Yaskawa INFORM job: N_R2_D34(P)(-165,-90).JBI

/JOB
//NAME N_R2_D34(P)(-165,-90)
//POS
///NPOS 212,212,212,10,0,0
///TOOL 0
///POSTYPE PULSE
///PULSE
C00000=-39723,-76225,-106677,19950,71807,76871
C00001=-136716,-73683,-105524,19345,72156,77265
C00002=-161407,-91524,-110310,15012,103390,71507
C00003=-108598,-106188,-63612,3932,70077,81231
C00004=-108146,-105032,-58861,3973,67731,81309
C00005=-107957,-104486,-56911,3991,66805,81343
C00006=-107899,-103124,-54603,4010,66084,81338
C00007=-107918,-103337,-55008,4006,66224,81336
C00008=-107946,-103390,-55013,4008,66201,81326
C00009=-107540,-105489,-55732,4011,65548,81444
C00010=-107946,-103390,-55013,4008,66201,81326
C00011=-108136,-103965,-56983,3989,67125,81292
C00012=-108589,-105196,-61782,3946,69462,81214
C00013=-104387,-140393,-91773,2539,65045,84360
C00014=-108543,-122383,-87788,3041,71761,81393
C00015=-108190,-121281,-83186,3043,69485,81459
C00016=-108044,-120747,-81302,3044,68596,81488
C00017=-107986,-119544,-79172,3051,67902,81491
C00018=-108002,-119703,-79496,3051,68020,81488
C00019=-108060,-119698,-79501,3057,68028,81468
C00020=-107657,-122309,-80316,3030,67174,81589
C00021=-108060,-119698,-79501,3057,68028,81468
C00022=-108206,-120261,-81401,3055,68912,81439
C00023=-108559,-121443,-86043,3052,71171,81373
C00024=-104043,-152650,-104301,-20,47297,80621
C00025=-107961,-134888,-100622,1830,53982,78996
C00026=-108046,-130238,-95035,1891,52935,78942
C00027=-108079,-128417,-92795,1916,52493,78920
C00028=-108021,-127286,-90730,1909,51803,78931
C00029=-108035,-127446,-91054,1912,51920,78927
C00030=-108130,-127490,-91067,1954,51908,78887
C00031=-107729,-130486,-91965,1802,50912,79038
C00032=-108130,-127490,-91067,1954,51908,78887
C00033=-108097,-129313,-93314,1928,52353,78910
C00034=-108012,-133964,-98916,1865,53408,78964
C00035=-177548,-171463,-116071,22976,53227,57999
C00036=-173065,-131414,-104138,1882,83052,64081
C00037=-174658,-131451,-100095,1929,80584,63502
C00038=-175319,-131311,-98421,1949,79642,63262
C00039=-175466,-130194,-96381,1956,78964,63202
C00040=-175319,-131311,-98421,1949,79642,63262
C00041=-175487,-130273,-96656,1956,79094,63196
C00042=-177055,-132761,-97424,1996,78327,62650
C00043=-175487,-130273,-96656,1956,79094,63196
C00044=-174824,-130456,-98346,1936,80024,63437
C00045=-173224,-130544,-102436,1888,82455,64018
C00046=-183578,-145461,-102579,23161,59534,56897
C00047=-173554,-122008,-87484,5289,73895,63503
C00048=-174753,-120461,-82756,5436,71868,62996
C00049=-175245,-119759,-80826,5498,71077,62789
C00050=-175392,-118530,-78687,5530,70405,62707
C00051=-175367,-118686,-78973,5525,70498,62719
C00052=-175370,-118724,-79021,5525,70509,62719
C00053=-176937,-120728,-79681,5662,69994,62147
C00054=-175370,-118724,-79021,5525,70509,62719
C00055=-174875,-119452,-80967,5462,71295,62928
C00056=-173672,-121073,-85733,5313,73308,63437
C00057=-178684,-130472,-89403,5463,71088,61622
C00058=-172855,-106156,-63418,1950,70986,63967
C00059=-174444,-104513,-58519,2015,68854,63388
C00060=-175103,-103777,-56512,2042,68014,63147
C00061=-175249,-102388,-54194,2055,67305,63085
C00062=-175217,-102613,-54582,2053,67427,63098
C00063=-175253,-102649,-54567,2054,67400,63085
C00064=-176818,-104272,-55156,2098,66967,62541
C00065=-175253,-102649,-54567,2054,67400,63085
C00066=-174591,-103412,-56593,2026,68239,63327
C00067=-172994,-105125,-61540,1961,70363,63910
C00068=-156260,-82084,-105549,20460,72443,69801
C00069=-137260,-84248,-120477,10166,77039,76481
C00070=-137260,-138866,-129024,10166,31486,76481
C00071=-31464,-162597,-129024,10166,12061,76481
C00072=11401,-148032,-125424,11666,35639,75770
C00073=126224,-114648,-117374,36487,17100,65054
C00074=135046,-120043,-103653,15284,86568,49617
C00075=106845,-105753,-62932,583,70286,77102
C00076=106393,-104585,-58171,607,67960,76935
C00077=106203,-104034,-56217,618,67041,76865
C00078=106162,-102674,-53905,622,66318,76847
C00079=106166,-102878,-54243,622,66421,76849
C00080=106334,-102921,-54287,616,66425,76907
C00081=105882,-105004,-55005,634,65800,76748
C00082=106334,-102921,-54287,616,66425,76907
C00083=106522,-103500,-56261,605,67341,76976
C00084=106972,-104744,-61071,581,69658,77143
C00085=104601,-139074,-91382,1569,66028,76192
C00086=106568,-121926,-87059,1557,71993,76932
C00087=106224,-120810,-82448,1613,69736,76782
C00088=106082,-120272,-80560,1636,68854,76720
C00089=106040,-119071,-78428,1648,68159,76695
C00090=106046,-119261,-78757,1646,68265,76699
C00091=106190,-119319,-78791,1631,68253,76749
C00092=105732,-121900,-79600,1688,67434,76576
C00093=106190,-119319,-78791,1631,68253,76749
C00094=106332,-119888,-80695,1608,69129,76811
C00095=106675,-121089,-85348,1552,71368,76961
C00096=103496,-155225,-104630,7919,46945,74289
C00097=105785,-134375,-99806,6437,54295,75766
C00098=105945,-129762,-94221,6456,53222,75764
C00099=106008,-127954,-91981,6467,52771,75762
C00100=105966,-126823,-89914,6544,52087,75701
C00101=105978,-126937,-90184,6529,52194,75712
C00102=106125,-127008,-90229,6468,52174,75772
C00103=105664,-129959,-91118,6752,51247,75517
C00104=106125,-127008,-90229,6468,52174,75772
C00105=106062,-128819,-92476,6456,52628,75775
C00106=105903,-133434,-98077,6434,53709,75777
C00107=128132,-113142,-93523,-3473,64221,79775
C00108=127541,-110622,-88467,-3323,62383,79607
C00109=127305,-109564,-86417,-3263,61656,79539
C00110=127138,-106637,-85321,-3181,62477,79452
C00111=127288,-110024,-87846,-3238,62297,79514
C00112=123322,-109914,-86529,-1878,61418,78027
C00113=118008,-109912,-86522,-16,61352,76001
C00114=114024,-109560,-86400,1379,61491,74484
C00115=114240,-110677,-88470,1295,62187,74574
C00116=114784,-113359,-93579,1090,63945,74797
C00117=120605,-145695,-100878,-6504,46630,80491
C00118=128077,-118688,-85011,-1726,71284,79523
C00119=126726,-104779,-76666,-1004,79571,78924
C00120=126488,-104947,-74265,-1002,78005,78856
C00121=126338,-102371,-73283,-996,78722,78799
C00122=126472,-105599,-75792,-1000,78609,78846
C00123=122432,-105195,-74343,-890,77878,77473
C00124=117012,-105110,-74308,-735,77846,75625
C00125=112968,-104735,-74177,-617,77924,74245
C00126=113438,-104642,-76602,-628,79468,74397
C00127=113371,-116037,-84290,-102,73201,74367
C00128=120594,-140938,-90128,-5435,60827,78775
C00129=125790,-88282,-54907,-1855,89205,80575
C00130=125481,-89790,-51762,-1908,86488,80513
C00131=125349,-90285,-50434,-1932,85415,80486
C00132=125231,-88136,-49532,-1951,85961,80439
C00133=125335,-91126,-52116,-1933,86017,80473
C00134=121365,-90427,-50480,-2603,85262,79186
C00135=116055,-90283,-50421,-3488,85105,77452
C00136=119868,-90564,-50050,-7604,84693,77985
C00137=120335,-90112,-51383,-7520,85779,78074
C00138=121427,-88708,-54542,-7332,88521,78274
C00139=128084,-118876,-109490,15608,91937,64784
C00140=126224,-114648,-117374,36487,17100,65054
C00141=118781,-153852,-129024,32591,23356,65054
C00142=12469,-167082,-125424,11666,16324,75770
C00143=-137258,-84249,-120477,10166,64820,76481
C00144=-160540,-100856,-113062,23154,68828,67580
C00145=-129704,-123203,-96216,9710,57100,77822
C00146=-128351,-111854,-90022,8241,62769,78816
C00147=-127965,-110264,-86953,8187,61668,78883
C00148=-127962,-110732,-88383,8139,62302,78931
C00149=-127784,-107324,-85860,8064,62480,79012
C00150=-123964,-110663,-87100,6807,61182,80388
C00151=-118738,-110727,-87139,4953,60792,82376
C00152=-114730,-110424,-87053,3503,60683,83913
C00153=-115087,-112114,-90154,3597,61737,83810
C00154=-115034,-127353,-96665,3487,52332,83552
C00155=-120587,-140955,-100514,6147,49960,81085
C00156=-130219,-122449,-86471,8825,68877,76131
C00157=-128194,-104501,-77199,7275,80206,77627
C00158=-127952,-104717,-74821,7301,78623,77617
C00159=-127948,-105352,-76341,7288,79227,77654
C00160=-127769,-102129,-73832,7281,79322,77721
C00161=-123925,-105065,-74954,7196,78166,78974
C00162=-118667,-105119,-74990,7025,77701,80756
C00163=-114634,-104852,-74915,6870,77446,82130
C00164=-115105,-104718,-77320,6855,79024,82055
C00165=-115436,-113024,-84089,6687,75142,81750
C00166=-120582,-141029,-90717,5476,61131,81670
C00167=-128285,-87656,-54320,10457,89548,79035
C00168=-127487,-89201,-51235,10596,86798,79071
C00169=-127146,-89710,-49931,10663,85708,79092
C00170=-127144,-90552,-51616,10658,86302,79143
C00171=-126986,-87570,-49030,10686,86223,79189
C00172=-123182,-89955,-50036,11339,85127,80359
C00173=-118012,-89954,-50056,12180,84414,82017
C00174=-114050,-89707,-49981,12789,83904,83291
C00175=-114638,-89281,-51315,12685,85009,83208
C00176=-116016,-87939,-54478,12458,87793,83023
C00177=-137088,-110527,-71299,-11812,85392,74901
C00178=-151248,-92745,-56294,-13309,83013,70315
C00179=-153775,-93208,-52742,-13646,80246,69760
C00180=-154842,-93280,-51259,-13793,79148,69522
C00181=-153977,-91331,-50464,-13683,79788,69743
C00182=-154783,-94178,-52960,-13764,79728,69477
C00183=-158502,-91409,-50586,-14135,79075,68289
C00184=-162995,-88717,-49588,-14508,79057,66760
C00185=-166247,-86464,-48726,-14744,79098,65642
C00186=-165114,-86470,-50212,-14620,80180,65901
C00187=-162400,-86203,-53771,-14331,82909,66512
C00188=-168399,-109053,-82349,-2367,78378,65064
C00189=-153094,-88623,-71084,-2982,100007,61638
C00190=-154899,-90939,-68502,-3287,97162,61087
C00191=-155658,-91729,-67395,-3417,96045,60858
C00192=-154888,-89489,-66414,-3281,96623,61105
C00193=-155605,-92249,-68886,-3413,96696,60858
C00194=-158825,-89499,-66505,-3999,96496,59762
C00195=-162743,-86354,-65215,-4713,97104,58398
C00196=-165600,-83764,-64121,-5229,97582,57396
C00197=-164765,-83025,-65209,-5099,98681,57638
C00198=-162766,-80848,-67746,-4792,101474,58222
C00199=-167065,-111844,-93662,10716,66234,64857
C00200=-163867,-82906,-82329,-2559,109140,68035
C00201=-165085,-87347,-80821,-2728,105894,67672
C00202=-165597,-88966,-80125,-2801,104618,67519
C00203=-165533,-89090,-81425,-2801,105355,67525
C00204=-164697,-86621,-79049,-2646,105191,67825
C00205=-162740,-91967,-81360,-2276,103927,68542
C00206=-158823,-95635,-82824,-1559,103037,69935
C00207=-155656,-98251,-83839,-981,102367,71052
C00208=-155268,-96625,-84596,-916,103674,71178
C00209=-154353,-92138,-86254,-764,107009,71479
C00210=-136716,-73683,-105524,19345,72156,77265
C00211=-39723,-76225,-106677,19950,71807,76871
BC00000=295325,674563,1075175
BC00001=353535,895977,1075175
BC00002=353535,975867,1075175
BC00003=342454,1030449,1075175
BC00004=342454,1030449,1075175
BC00005=342454,1030449,1075175
BC00006=342454,1030449,1075175
BC00007=342454,1030449,1075175
BC00008=342454,1030449,1075175
BC00009=342454,1030449,1075175
BC00010=342454,1030449,1075175
BC00011=342454,1030449,1075175
BC00012=342454,1030449,1075175
BC00013=342372,1053588,1075175
BC00014=342372,1053588,1075175
BC00015=342372,1053588,1075175
BC00016=342372,1053588,1075175
BC00017=342372,1053588,1075175
BC00018=342372,1053588,1075175
BC00019=342372,1053588,1075175
BC00020=342372,1053588,1075175
BC00021=342372,1053588,1075175
BC00022=342372,1053588,1075175
BC00023=342372,1053588,1075175
BC00024=339313,1046331,1075175
BC00025=339313,1046331,1075175
BC00026=339313,1046331,1075175
BC00027=339313,1046331,1075175
BC00028=339313,1046331,1075175
BC00029=339313,1046331,1075175
BC00030=339313,1046331,1075175
BC00031=339313,1046331,1075175
BC00032=339313,1046331,1075175
BC00033=339313,1046331,1075175
BC00034=339313,1046331,1075175
BC00035=316444,1061550,1075175
BC00036=316336,1108016,1075175
BC00037=316336,1108016,1075175
BC00038=316336,1108016,1075175
BC00039=316336,1108016,1075175
BC00040=316336,1108016,1075175
BC00041=316336,1108016,1075175
BC00042=316336,1108016,1075175
BC00043=316336,1108016,1075175
BC00044=316336,1108016,1075175
BC00045=316336,1108016,1075175
BC00046=316444,1061550,1075175
BC00047=316378,1069449,1075175
BC00048=316378,1069449,1075175
BC00049=316378,1069449,1075175
BC00050=316378,1069449,1075175
BC00051=316378,1069449,1075175
BC00052=316378,1069449,1075175
BC00053=316378,1069449,1075175
BC00054=316378,1069449,1075175
BC00055=316378,1069449,1075175
BC00056=316378,1069449,1075175
BC00057=316378,1069449,1075175
BC00058=316510,1046311,1075175
BC00059=316510,1046311,1075175
BC00060=316510,1046311,1075175
BC00061=316510,1046311,1075175
BC00062=316510,1046311,1075175
BC00063=316510,1046311,1075175
BC00064=316510,1046311,1075175
BC00065=316510,1046311,1075175
BC00066=316510,1046311,1075175
BC00067=316510,1046311,1075175
BC00068=381896,966588,1075175
BC00069=353816,923989,1075175
BC00070=353816,923989,1075175
BC00071=379773,1126391,1075175
BC00072=398190,1030285,1075175
BC00073=312632,1138057,1075175
BC00074=340753,1115300,1075175
BC00075=348057,1094074,1075175
BC00076=348057,1094074,1075175
BC00077=348057,1094074,1075175
BC00078=348057,1094074,1075175
BC00079=348057,1094074,1075175
BC00080=348057,1094074,1075175
BC00081=348057,1094074,1075175
BC00082=348057,1094074,1075175
BC00083=348057,1094074,1075175
BC00084=348057,1094074,1075175
BC00085=347868,1070766,1075175
BC00086=347868,1070766,1075175
BC00087=347868,1070766,1075175
BC00088=347868,1070766,1075175
BC00089=347868,1070766,1075175
BC00090=347868,1070766,1075175
BC00091=347868,1070766,1075175
BC00092=347868,1070766,1075175
BC00093=347868,1070766,1075175
BC00094=347868,1070766,1075175
BC00095=347868,1070766,1075175
BC00096=347977,1078609,1075175
BC00097=347977,1078609,1075175
BC00098=347977,1078609,1075175
BC00099=347977,1078609,1075175
BC00100=347977,1078609,1075175
BC00101=347977,1078609,1075175
BC00102=347977,1078609,1075175
BC00103=347977,1078609,1075175
BC00104=347977,1078609,1075175
BC00105=347977,1078609,1075175
BC00106=347977,1078609,1075175
BC00107=359186,1090753,1075175
BC00108=359186,1090753,1075175
BC00109=359186,1090753,1075175
BC00110=359186,1090753,1075175
BC00111=359186,1090753,1075175
BC00112=359186,1090753,1075175
BC00113=359186,1090753,1075175
BC00114=359186,1090753,1075175
BC00115=359186,1090753,1075175
BC00116=359186,1090753,1075175
BC00117=343034,1090568,1075175
BC00118=358057,1077191,1075175
BC00119=358057,1077191,1075175
BC00120=358057,1077191,1075175
BC00121=358057,1077191,1075175
BC00122=358057,1077191,1075175
BC00123=358057,1077191,1075175
BC00124=358057,1077191,1075175
BC00125=358057,1077191,1075175
BC00126=358057,1077191,1075175
BC00127=358057,1077191,1075175
BC00128=343077,1074128,1075175
BC00129=353730,1083739,1057896
BC00130=353730,1083739,1057896
BC00131=353730,1083739,1057896
BC00132=353730,1083739,1057896
BC00133=353730,1083739,1057896
BC00134=353730,1083739,1057896
BC00135=353730,1083739,1057896
BC00136=353730,1083739,1057896
BC00137=353730,1083739,1057896
BC00138=353730,1083739,1057896
BC00139=340753,1115300,1075175
BC00140=312632,1138057,1075175
BC00141=312632,1138057,1075175
BC00142=398190,1030285,1075175
BC00143=353817,923990,1075175
BC00144=381896,966588,1075175
BC00145=352359,1033679,1075175
BC00146=352359,1033679,1075175
BC00147=352359,1033679,1075175
BC00148=352359,1033679,1075175
BC00149=352359,1033679,1075175
BC00150=352359,1033679,1075175
BC00151=352359,1033679,1075175
BC00152=352359,1033679,1075175
BC00153=352359,1033679,1075175
BC00154=352359,1033679,1075175
BC00155=343481,1033212,1075175
BC00156=349388,1046228,1075175
BC00157=349388,1046228,1075175
BC00158=349388,1046228,1075175
BC00159=349388,1046228,1075175
BC00160=349388,1046228,1075175
BC00161=349388,1046228,1075175
BC00162=349388,1046228,1075175
BC00163=349388,1046228,1075175
BC00164=349388,1046228,1075175
BC00165=349388,1046228,1075175
BC00166=343531,1049804,1075175
BC00167=339512,1039360,1057640
BC00168=339512,1039360,1057640
BC00169=339512,1039360,1057640
BC00170=339512,1039360,1057640
BC00171=339512,1039360,1057640
BC00172=339512,1039360,1057640
BC00173=339512,1039360,1057640
BC00174=339512,1039360,1057640
BC00175=339512,1039360,1057640
BC00176=339512,1039360,1057640
BC00177=341311,1059119,1075175
BC00178=330413,1051315,1057925
BC00179=330413,1051315,1057925
BC00180=330413,1051315,1057925
BC00181=330413,1051315,1057925
BC00182=330413,1051315,1057925
BC00183=330413,1051315,1057925
BC00184=330413,1051315,1057925
BC00185=330413,1051315,1057925
BC00186=330413,1051315,1057925
BC00187=330413,1051315,1057925
BC00188=337538,1050257,1075175
BC00189=315681,1075300,1075175
BC00190=315681,1075300,1075175
BC00191=315681,1075300,1075175
BC00192=315681,1075300,1075175
BC00193=315681,1075300,1075175
BC00194=315681,1075300,1075175
BC00195=315681,1075300,1075175
BC00196=315681,1075300,1075175
BC00197=315681,1075300,1075175
BC00198=315681,1075300,1075175
BC00199=337544,1033689,1075175
BC00200=308612,1102150,1075175
BC00201=308612,1102150,1075175
BC00202=308612,1102150,1075175
BC00203=308612,1102150,1075175
BC00204=308612,1102150,1075175
BC00205=308612,1102150,1075175
BC00206=308612,1102150,1075175
BC00207=308612,1102150,1075175
BC00208=308612,1102150,1075175
BC00209=308612,1102150,1075175
BC00210=353535,895977,1075175
BC00211=295325,674563,1075175
EC00000=-1463287,-556475
EC00001=-1463287,-556475
EC00002=-1463287,-556475
EC00003=-1463287,-556475
EC00004=-1463287,-556475
EC00005=-1463287,-556475
EC00006=-1463287,-556475
EC00007=-1463287,-556475
EC00008=-1463287,-556475
EC00009=-1463287,-556475
EC00010=-1463287,-556475
EC00011=-1463287,-556475
EC00012=-1463287,-556475
EC00013=-1463287,-556475
EC00014=-1463287,-556475
EC00015=-1463287,-556475
EC00016=-1463287,-556475
EC00017=-1463287,-556475
EC00018=-1463287,-556475
EC00019=-1463287,-556475
EC00020=-1463287,-556475
EC00021=-1463287,-556475
EC00022=-1463287,-556475
EC00023=-1463287,-556475
EC00024=-1463287,-556475
EC00025=-1463287,-556475
EC00026=-1463287,-556475
EC00027=-1463287,-556475
EC00028=-1463287,-556475
EC00029=-1463287,-556475
EC00030=-1463287,-556475
EC00031=-1463287,-556475
EC00032=-1463287,-556475
EC00033=-1463287,-556475
EC00034=-1463287,-556475
EC00035=-1463287,-556475
EC00036=-1463287,-556475
EC00037=-1463287,-556475
EC00038=-1463287,-556475
EC00039=-1463287,-556475
EC00040=-1463287,-556475
EC00041=-1463287,-556475
EC00042=-1463287,-556475
EC00043=-1463287,-556475
EC00044=-1463287,-556475
EC00045=-1463287,-556475
EC00046=-1463287,-556475
EC00047=-1463287,-556475
EC00048=-1463287,-556475
EC00049=-1463287,-556475
EC00050=-1463287,-556475
EC00051=-1463287,-556475
EC00052=-1463287,-556475
EC00053=-1463287,-556475
EC00054=-1463287,-556475
EC00055=-1463287,-556475
EC00056=-1463287,-556475
EC00057=-1463287,-556475
EC00058=-1463287,-556475
EC00059=-1463287,-556475
EC00060=-1463287,-556475
EC00061=-1463287,-556475
EC00062=-1463287,-556475
EC00063=-1463287,-556475
EC00064=-1463287,-556475
EC00065=-1463287,-556475
EC00066=-1463287,-556475
EC00067=-1463287,-556475
EC00068=-1463287,-556475
EC00069=-1463287,-556475
EC00070=-1463287,-556475
EC00071=-1463287,-556475
EC00072=-1595090,-3837
EC00073=-1729339,556475
EC00074=-1729339,556475
EC00075=-1729339,556475
EC00076=-1729339,556475
EC00077=-1729339,556475
EC00078=-1729339,556475
EC00079=-1729339,556475
EC00080=-1729339,556475
EC00081=-1729339,556475
EC00082=-1729339,556475
EC00083=-1729339,556475
EC00084=-1729339,556475
EC00085=-1729339,556475
EC00086=-1729339,556475
EC00087=-1729339,556475
EC00088=-1729339,556475
EC00089=-1729339,556475
EC00090=-1729339,556475
EC00091=-1729339,556475
EC00092=-1729339,556475
EC00093=-1729339,556475
EC00094=-1729339,556475
EC00095=-1729339,556475
EC00096=-1729339,556475
EC00097=-1729339,556475
EC00098=-1729339,556475
EC00099=-1729339,556475
EC00100=-1729339,556475
EC00101=-1729339,556475
EC00102=-1729339,556475
EC00103=-1729339,556475
EC00104=-1729339,556475
EC00105=-1729339,556475
EC00106=-1729339,556475
EC00107=-1729339,556475
EC00108=-1729339,556475
EC00109=-1729339,556475
EC00110=-1729339,556475
EC00111=-1729339,556475
EC00112=-1729339,556475
EC00113=-1729339,556475
EC00114=-1729339,556475
EC00115=-1729339,556475
EC00116=-1729339,556475
EC00117=-1729339,556475
EC00118=-1729339,556475
EC00119=-1729339,556475
EC00120=-1729339,556475
EC00121=-1729339,556475
EC00122=-1729339,556475
EC00123=-1729339,556475
EC00124=-1729339,556475
EC00125=-1729339,556475
EC00126=-1729339,556475
EC00127=-1729339,556475
EC00128=-1729339,556475
EC00129=-1729339,556475
EC00130=-1729339,556475
EC00131=-1729339,556475
EC00132=-1729339,556475
EC00133=-1729339,556475
EC00134=-1729339,556475
EC00135=-1729339,556475
EC00136=-1729339,556475
EC00137=-1729339,556475
EC00138=-1729339,556475
EC00139=-1729339,556475
EC00140=-1729339,556475
EC00141=-1729339,556475
EC00142=-1595090,-3837
EC00143=-1463287,-556475
EC00144=-1463287,-556475
EC00145=-1463287,-556475
EC00146=-1463287,-556475
EC00147=-1463287,-556475
EC00148=-1463287,-556475
EC00149=-1463287,-556475
EC00150=-1463287,-556475
EC00151=-1463287,-556475
EC00152=-1463287,-556475
EC00153=-1463287,-556475
EC00154=-1463287,-556475
EC00155=-1463287,-556475
EC00156=-1463287,-556475
EC00157=-1463287,-556475
EC00158=-1463287,-556475
EC00159=-1463287,-556475
EC00160=-1463287,-556475
EC00161=-1463287,-556475
EC00162=-1463287,-556475
EC00163=-1463287,-556475
EC00164=-1463287,-556475
EC00165=-1463287,-556475
EC00166=-1463287,-556475
EC00167=-1463287,-556475
EC00168=-1463287,-556475
EC00169=-1463287,-556475
EC00170=-1463287,-556475
EC00171=-1463287,-556475
EC00172=-1463287,-556475
EC00173=-1463287,-556475
EC00174=-1463287,-556475
EC00175=-1463287,-556475
EC00176=-1463287,-556475
EC00177=-1463287,-556475
EC00178=-1463287,-556475
EC00179=-1463287,-556475
EC00180=-1463287,-556475
EC00181=-1463287,-556475
EC00182=-1463287,-556475
EC00183=-1463287,-556475
EC00184=-1463287,-556475
EC00185=-1463287,-556475
EC00186=-1463287,-556475
EC00187=-1463287,-556475
EC00188=-1463287,-556475
EC00189=-1463287,-556475
EC00190=-1463287,-556475
EC00191=-1463287,-556475
EC00192=-1463287,-556475
EC00193=-1463287,-556475
EC00194=-1463287,-556475
EC00195=-1463287,-556475
EC00196=-1463287,-556475
EC00197=-1463287,-556475
EC00198=-1463287,-556475
EC00199=-1463287,-556475
EC00200=-1463287,-556475
EC00201=-1463287,-556475
EC00202=-1463287,-556475
EC00203=-1463287,-556475
EC00204=-1463287,-556475
EC00205=-1463287,-556475
EC00206=-1463287,-556475
EC00207=-1463287,-556475
EC00208=-1463287,-556475
EC00209=-1463287,-556475
EC00210=-1463287,-556475
EC00211=-1463287,-556475
///POSTYPE BASE
///RECTAN
///RCONF 0,0,0,0,0,0,0,0,0,0,0,0,0,0,0,0,0,0,0,0,0,0,0,0
P00006=0.222,-3.123,-1.508,0.0000,0.0000,0.0000
P00021=-0.225,-6.128,-0.405,0.0000,0.0000,0.0000
P00022=0.222,-3.123,-1.508,0.0000,0.0000,0.0000
P00023=0.143,-0.036,0.682,0.0000,0.0000,0.0000
P00024=0.145,-0.552,1.326,0.0000,0.0000,0.0000
P00025=-2.003,0.006,0.728,0.0000,0.0000,0.0000
P00026=0.562,-0.002,-0.337,0.0000,0.0000,0.0000
P00034=-0.304,0.773,-2.693,0.0000,0.0000,0.0000
P00035=2.817,0.591,-1.622,0.0000,0.0000,0.0000
P00036=-1.108,-0.829,1.850,0.0000,0.0000,0.0000
//INST
///DATE 2024/02/02 10:05
///ATTR SC,RW
///GROUP1 RB1,BS1
///GROUP2 ST1
NOP
'N_r2_D34(P)(-165,-90)
MOVJ C00000 BC00000 VJ=100.00  +MOVJ EC00000 VJ=100.00
MOVJ C00001 BC00001 VJ=100.00  +MOVJ EC00001 VJ=100.00
MOVJ C00002 BC00002 VJ=100.00  +MOVJ EC00002 VJ=100.00
'Path S3213
SSFTOF
MOVJ C00003 BC00003 VJ=100.00  +MOVJ EC00003 VJ=100.00
MOVL C00004 BC00004 V=400.0  +MOVJ EC00004 VJ=100.00
SMOVL C00005 BC00005 V=60.0  +MOVJ EC00005
SREFP 3 C00006 BC00006  +REFP EC00006
CALL JOB:SEARCH-R1-S1
SET P021 P006
SSFTON P021
SMOVL C00007 BC00007 V=60.0  +MOVJ EC00007
SMOVL C00008 BC00008 V=60.0  +MOVJ EC00008
SREFP 3 C00009 BC00009  +REFP EC00009
CALL JOB:SEARCH-R1-S1
SET P021 P006
SSFTON P021
SMOVL C00010 BC00010 V=60.0  +MOVJ EC00010
MOVL C00011 BC00011 V=400.0  +MOVJ EC00011 VJ=100.00
MOVL C00012 BC00012 V=1000.0  +MOVJ EC00012 VJ=100.00
MOVJ C00013 BC00013 VJ=100.00  +MOVJ EC00013 VJ=100.00
'Path S3214
SSFTOF
MOVJ C00014 BC00014 VJ=100.00  +MOVJ EC00014 VJ=100.00
MOVL C00015 BC00015 V=400.0  +MOVJ EC00015 VJ=100.00
SMOVL C00016 BC00016 V=60.0  +MOVJ EC00016
SREFP 3 C00017 BC00017  +REFP EC00017
CALL JOB:SEARCH-R1-S1
SET P022 P006
SSFTON P022
SMOVL C00018 BC00018 V=60.0  +MOVJ EC00018
SMOVL C00019 BC00019 V=60.0  +MOVJ EC00019
SREFP 3 C00020 BC00020  +REFP EC00020
CALL JOB:SEARCH-R1-S1
SET P022 P006
SSFTON P022
SMOVL C00021 BC00021 V=60.0  +MOVJ EC00021
MOVL C00022 BC00022 V=400.0  +MOVJ EC00022 VJ=100.00
MOVL C00023 BC00023 V=1000.0  +MOVJ EC00023 VJ=100.00
MOVJ C00024 BC00024 VJ=100.00  +MOVJ EC00024 VJ=100.00
'Path S3215
SSFTOF
MOVJ C00025 BC00025 VJ=100.00  +MOVJ EC00025 VJ=100.00
MOVL C00026 BC00026 V=400.0  +MOVJ EC00026 VJ=100.00
SMOVL C00027 BC00027 V=60.0  +MOVJ EC00027
SREFP 3 C00028 BC00028  +REFP EC00028
CALL JOB:SEARCH-R1-S1
SET P023 P006
SSFTON P023
SMOVL C00029 BC00029 V=60.0  +MOVJ EC00029
SMOVL C00030 BC00030 V=60.0  +MOVJ EC00030
SREFP 3 C00031 BC00031  +REFP EC00031
CALL JOB:SEARCH-R1-S1
SET P023 P006
SSFTON P023
SMOVL C00032 BC00032 V=60.0  +MOVJ EC00032
MOVL C00033 BC00033 V=400.0  +MOVJ EC00033 VJ=100.00
MOVL C00034 BC00034 V=1000.0  +MOVJ EC00034 VJ=100.00
MOVJ C00035 BC00035 VJ=100.00  +MOVJ EC00035 VJ=100.00
'Path S3216
SSFTOF
MOVJ C00036 BC00036 VJ=100.00  +MOVJ EC00036 VJ=100.00
MOVL C00037 BC00037 V=400.0  +MOVJ EC00037 VJ=100.00
SMOVL C00038 BC00038 V=60.0  +MOVJ EC00038
SREFP 3 C00039 BC00039  +REFP EC00039
CALL JOB:SEARCH-R1-S1
SET P024 P006
SSFTON P024
SMOVL C00040 BC00040 V=60.0  +MOVJ EC00040
SMOVL C00041 BC00041 V=60.0  +MOVJ EC00041
SREFP 3 C00042 BC00042  +REFP EC00042
CALL JOB:SEARCH-R1-S1
SET P024 P006
SSFTON P024
SMOVL C00043 BC00043 V=60.0  +MOVJ EC00043
MOVL C00044 BC00044 V=400.0  +MOVJ EC00044 VJ=100.00
MOVL C00045 BC00045 V=1000.0  +MOVJ EC00045 VJ=100.00
MOVJ C00046 BC00046 VJ=100.00  +MOVJ EC00046 VJ=100.00
'Path S3217
SSFTOF
MOVJ C00047 BC00047 VJ=100.00  +MOVJ EC00047 VJ=100.00
MOVL C00048 BC00048 V=400.0  +MOVJ EC00048 VJ=100.00
SMOVL C00049 BC00049 V=60.0  +MOVJ EC00049
SREFP 3 C00050 BC00050  +REFP EC00050
CALL JOB:SEARCH-R1-S1
SET P025 P006
SSFTON P025
SMOVL C00051 BC00051 V=60.0  +MOVJ EC00051
SMOVL C00052 BC00052 V=60.0  +MOVJ EC00052
SREFP 3 C00053 BC00053  +REFP EC00053
CALL JOB:SEARCH-R1-S1
SET P025 P006
SSFTON P025
SMOVL C00054 BC00054 V=60.0  +MOVJ EC00054
MOVL C00055 BC00055 V=400.0  +MOVJ EC00055 VJ=100.00
MOVL C00056 BC00056 V=1000.0  +MOVJ EC00056 VJ=100.00
MOVJ C00057 BC00057 VJ=100.00  +MOVJ EC00057 VJ=100.00
'Path S3218
SSFTOF
MOVJ C00058 BC00058 VJ=100.00  +MOVJ EC00058 VJ=100.00
MOVL C00059 BC00059 V=400.0  +MOVJ EC00059 VJ=100.00
SMOVL C00060 BC00060 V=60.0  +MOVJ EC00060
SREFP 3 C00061 BC00061  +REFP EC00061
CALL JOB:SEARCH-R1-S1
SET P026 P006
SSFTON P026
SMOVL C00062 BC00062 V=60.0  +MOVJ EC00062
SMOVL C00063 BC00063 V=60.0  +MOVJ EC00063
SREFP 3 C00064 BC00064  +REFP EC00064
CALL JOB:SEARCH-R1-S1
SET P026 P006
SSFTON P026
SMOVL C00065 BC00065 V=60.0  +MOVJ EC00065
MOVL C00066 BC00066 V=400.0  +MOVJ EC00066 VJ=100.00
MOVL C00067 BC00067 V=1000.0  +MOVJ EC00067 VJ=100.00
'obrot
MOVJ C00068 BC00068 VJ=100.00  +MOVJ EC00068 VJ=100.00
MOVJ C00069 BC00069 VJ=100.00  +MOVJ EC00069 VJ=100.00
MOVJ C00070 BC00070 VJ=100.00  +MOVJ EC00070 VJ=100.00
MOVJ C00071 BC00071 VJ=100.00  +MOVJ EC00071 VJ=100.00
MOVJ C00072 BC00072 VJ=100.00  +MOVJ EC00072 VJ=100.00
MOVJ C00073 BC00073 VJ=100.00  +MOVJ EC00073 VJ=100.00
MOVJ C00074 BC00074 VJ=100.00  +MOVJ EC00074 VJ=100.00
'
'Path S3219
SSFTOF
MOVJ C00075 BC00075 VJ=100.00  +MOVJ EC00075 VJ=100.00
MOVL C00076 BC00076 V=400.0  +MOVJ EC00076 VJ=100.00
SMOVL C00077 BC00077 V=60.0  +MOVJ EC00077
SREFP 3 C00078 BC00078  +REFP EC00078
CALL JOB:SEARCH-R1-S1
SET P034 P006
SSFTON P034
SMOVL C00079 BC00079 V=60.0  +MOVJ EC00079
SMOVL C00080 BC00080 V=60.0  +MOVJ EC00080
SREFP 3 C00081 BC00081  +REFP EC00081
CALL JOB:SEARCH-R1-S1
SET P034 P006
SSFTON P034
SMOVL C00082 BC00082 V=60.0  +MOVJ EC00082
MOVL C00083 BC00083 V=400.0  +MOVJ EC00083 VJ=100.00
MOVL C00084 BC00084 V=1000.0  +MOVJ EC00084 VJ=100.00
MOVJ C00085 BC00085 VJ=100.00  +MOVJ EC00085 VJ=100.00
'Path S3220
SSFTOF
MOVJ C00086 BC00086 VJ=100.00  +MOVJ EC00086 VJ=100.00
MOVL C00087 BC00087 V=400.0  +MOVJ EC00087 VJ=100.00
SMOVL C00088 BC00088 V=60.0  +MOVJ EC00088
SREFP 3 C00089 BC00089  +REFP EC00089
CALL JOB:SEARCH-R1-S1
SET P035 P006
SSFTON P035
SMOVL C00090 BC00090 V=60.0  +MOVJ EC00090
SMOVL C00091 BC00091 V=60.0  +MOVJ EC00091
SREFP 3 C00092 BC00092  +REFP EC00092
CALL JOB:SEARCH-R1-S1
SET P035 P006
SSFTON P035
SMOVL C00093 BC00093 V=60.0  +MOVJ EC00093
MOVL C00094 BC00094 V=400.0  +MOVJ EC00094 VJ=100.00
MOVL C00095 BC00095 V=1000.0  +MOVJ EC00095 VJ=100.00
MOVJ C00096 BC00096 VJ=100.00  +MOVJ EC00096 VJ=100.00
'Path S3221
SSFTOF
MOVJ C00097 BC00097 VJ=100.00  +MOVJ EC00097 VJ=100.00
MOVL C00098 BC00098 V=400.0  +MOVJ EC00098 VJ=100.00
SMOVL C00099 BC00099 V=60.0  +MOVJ EC00099
SREFP 3 C00100 BC00100  +REFP EC00100
CALL JOB:SEARCH-R1-S1
SET P036 P006
SSFTON P036
SMOVL C00101 BC00101 V=60.0  +MOVJ EC00101
SMOVL C00102 BC00102 V=60.0  +MOVJ EC00102
SREFP 3 C00103 BC00103  +REFP EC00103
CALL JOB:SEARCH-R1-S1
SET P036 P006
SSFTON P036
SMOVL C00104 BC00104 V=60.0  +MOVJ EC00104
MOVL C00105 BC00105 V=400.0  +MOVJ EC00105 VJ=100.00
MOVL C00106 BC00106 V=1000.0  +MOVJ EC00106 VJ=100.00
'Path W3222
SSFTOF
SSFTON P036
MOVJ C00107 BC00107 VJ=100.00  +MOVJ EC00107 VJ=100.00
SMOVL C00108 BC00108 V=400.0  +MOVJ EC00108
SMOVL C00109 BC00109 V=100.0 PL=0  +MOVJ EC00109
SREFP 1 C00110 BC00110  +REFP EC00110
SREFP 2 C00111 BC00111  +REFP EC00111
MACRO1 MJ#(0) ARGF0
ARCON
SMOVL C00112 BC00112 V=10.0  +MOVJ EC00112
SMOVL C00113 BC00113 V=10.0  +MOVJ EC00113
SMOVL C00114 BC00114 V=10.0  +MOVJ EC00114
ARCOF
SMOVL C00115 BC00115 V=400.0  +MOVJ EC00115
SMOVL C00116 BC00116 V=1000.0  +MOVJ EC00116
SSFTOF
MOVJ C00117 BC00117 VJ=100.00  +MOVJ EC00117 VJ=100.00
'Path W3223
SSFTOF
SSFTON P035
MOVJ C00118 BC00118 VJ=100.00  +MOVJ EC00118 VJ=100.00
SMOVL C00119 BC00119 V=400.0  +MOVJ EC00119
SMOVL C00120 BC00120 V=100.0 PL=0  +MOVJ EC00120
SREFP 1 C00121 BC00121  +REFP EC00121
SREFP 2 C00122 BC00122  +REFP EC00122
MACRO1 MJ#(0) ARGF0
ARCON
SMOVL C00123 BC00123 V=10.0  +MOVJ EC00123
SMOVL C00124 BC00124 V=10.0  +MOVJ EC00124
SMOVL C00125 BC00125 V=10.0  +MOVJ EC00125
ARCOF
SMOVL C00126 BC00126 V=400.0  +MOVJ EC00126
SMOVL C00127 BC00127 V=1000.0  +MOVJ EC00127
SSFTOF
MOVJ C00128 BC00128 VJ=100.00  +MOVJ EC00128 VJ=100.00
'Path W3224
SSFTOF
SSFTON P034
MOVJ C00129 BC00129 VJ=100.00  +MOVJ EC00129 VJ=100.00
SMOVL C00130 BC00130 V=400.0  +MOVJ EC00130
SMOVL C00131 BC00131 V=100.0 PL=0  +MOVJ EC00131
SREFP 1 C00132 BC00132  +REFP EC00132
SREFP 2 C00133 BC00133  +REFP EC00133
MACRO1 MJ#(0) ARGF0
ARCON
SMOVL C00134 BC00134 V=10.0  +MOVJ EC00134
SMOVL C00135 BC00135 V=10.0  +MOVJ EC00135
SMOVL C00136 BC00136 V=10.0  +MOVJ EC00136
ARCOF
SMOVL C00137 BC00137 V=400.0  +MOVJ EC00137
SMOVL C00138 BC00138 V=1000.0  +MOVJ EC00138
SSFTOF
'obrot
MOVJ C00139 BC00139 VJ=100.00  +MOVJ EC00139 VJ=100.00
MOVJ C00140 BC00140 VJ=100.00  +MOVJ EC00140 VJ=100.00
MOVJ C00141 BC00141 VJ=100.00  +MOVJ EC00141 VJ=100.00
MOVJ C00142 BC00142 VJ=100.00  +MOVJ EC00142 VJ=100.00
MOVJ C00143 BC00143 VJ=100.00  +MOVJ EC00143 VJ=100.00
MOVJ C00144 BC00144 VJ=100.00  +MOVJ EC00144 VJ=100.00
'
'Path W3225
SSFTOF
SSFTON P023
MOVJ C00145 BC00145 VJ=100.00  +MOVJ EC00145 VJ=100.00
SMOVL C00146 BC00146 V=400.0  +MOVJ EC00146
SMOVL C00147 BC00147 V=100.0 PL=0  +MOVJ EC00147
SREFP 1 C00148 BC00148  +REFP EC00148
SREFP 2 C00149 BC00149  +REFP EC00149
MACRO1 MJ#(0) ARGF0
ARCON
SMOVL C00150 BC00150 V=10.0  +MOVJ EC00150
SMOVL C00151 BC00151 V=10.0  +MOVJ EC00151
SMOVL C00152 BC00152 V=10.0  +MOVJ EC00152
ARCOF
SMOVL C00153 BC00153 V=400.0  +MOVJ EC00153
SMOVL C00154 BC00154 V=1000.0  +MOVJ EC00154
SSFTOF
MOVJ C00155 BC00155 VJ=100.00  +MOVJ EC00155 VJ=100.00
'Path W3226
SSFTOF
SSFTON P022
MOVJ C00156 BC00156 VJ=100.00  +MOVJ EC00156 VJ=100.00
SMOVL C00157 BC00157 V=400.0  +MOVJ EC00157
SMOVL C00158 BC00158 V=100.0 PL=0  +MOVJ EC00158
SREFP 1 C00159 BC00159  +REFP EC00159
SREFP 2 C00160 BC00160  +REFP EC00160
MACRO1 MJ#(0) ARGF0
ARCON
SMOVL C00161 BC00161 V=10.0  +MOVJ EC00161
SMOVL C00162 BC00162 V=10.0  +MOVJ EC00162
SMOVL C00163 BC00163 V=10.0  +MOVJ EC00163
ARCOF
SMOVL C00164 BC00164 V=400.0  +MOVJ EC00164
SMOVL C00165 BC00165 V=1000.0  +MOVJ EC00165
SSFTOF
MOVJ C00166 BC00166 VJ=100.00  +MOVJ EC00166 VJ=100.00
'Path W3227
SSFTOF
SSFTON P021
MOVJ C00167 BC00167 VJ=100.00  +MOVJ EC00167 VJ=100.00
SMOVL C00168 BC00168 V=400.0  +MOVJ EC00168
SMOVL C00169 BC00169 V=100.0 PL=0  +MOVJ EC00169
SREFP 1 C00170 BC00170  +REFP EC00170
SREFP 2 C00171 BC00171  +REFP EC00171
MACRO1 MJ#(0) ARGF0
ARCON
SMOVL C00172 BC00172 V=10.0  +MOVJ EC00172
SMOVL C00173 BC00173 V=10.0  +MOVJ EC00173
SMOVL C00174 BC00174 V=10.0  +MOVJ EC00174
ARCOF
SMOVL C00175 BC00175 V=400.0  +MOVJ EC00175
SMOVL C00176 BC00176 V=1000.0  +MOVJ EC00176
SSFTOF
MOVJ C00177 BC00177 VJ=100.00  +MOVJ EC00177 VJ=100.00
'Path W3228
SSFTOF
SSFTON P026
MOVJ C00178 BC00178 VJ=100.00  +MOVJ EC00178 VJ=100.00
SMOVL C00179 BC00179 V=400.0  +MOVJ EC00179
SMOVL C00180 BC00180 V=100.0 PL=0  +MOVJ EC00180
SREFP 1 C00181 BC00181  +REFP EC00181
SREFP 2 C00182 BC00182  +REFP EC00182
MACRO1 MJ#(0) ARGF0
ARCON
SMOVL C00183 BC00183 V=10.0  +MOVJ EC00183
SMOVL C00184 BC00184 V=10.0  +MOVJ EC00184
SMOVL C00185 BC00185 V=10.0  +MOVJ EC00185
ARCOF
SMOVL C00186 BC00186 V=400.0  +MOVJ EC00186
SMOVL C00187 BC00187 V=1000.0  +MOVJ EC00187
SSFTOF
MOVJ C00188 BC00188 VJ=100.00  +MOVJ EC00188 VJ=100.00
'Path W3229
SSFTOF
SSFTON P025
MOVJ C00189 BC00189 VJ=100.00  +MOVJ EC00189 VJ=100.00
SMOVL C00190 BC00190 V=400.0  +MOVJ EC00190
SMOVL C00191 BC00191 V=100.0 PL=0  +MOVJ EC00191
SREFP 1 C00192 BC00192  +REFP EC00192
SREFP 2 C00193 BC00193  +REFP EC00193
MACRO1 MJ#(0) ARGF0
ARCON
SMOVL C00194 BC00194 V=10.0  +MOVJ EC00194
SMOVL C00195 BC00195 V=10.0  +MOVJ EC00195
SMOVL C00196 BC00196 V=10.0  +MOVJ EC00196
ARCOF
SMOVL C00197 BC00197 V=400.0  +MOVJ EC00197
SMOVL C00198 BC00198 V=1000.0  +MOVJ EC00198
SSFTOF
MOVJ C00199 BC00199 VJ=100.00  +MOVJ EC00199 VJ=100.00
'Path W3230
SSFTOF
SSFTON P024
MOVJ C00200 BC00200 VJ=100.00  +MOVJ EC00200 VJ=100.00
SMOVL C00201 BC00201 V=400.0  +MOVJ EC00201
SMOVL C00202 BC00202 V=100.0 PL=0  +MOVJ EC00202
SREFP 1 C00203 BC00203  +REFP EC00203
SREFP 2 C00204 BC00204  +REFP EC00204
MACRO1 MJ#(0) ARGF0
ARCON
SMOVL C00205 BC00205 V=10.0  +MOVJ EC00205
SMOVL C00206 BC00206 V=10.0  +MOVJ EC00206
SMOVL C00207 BC00207 V=10.0  +MOVJ EC00207
ARCOF
SMOVL C00208 BC00208 V=400.0  +MOVJ EC00208
SMOVL C00209 BC00209 V=1000.0  +MOVJ EC00209
SSFTOF
MOVJ C00210 BC00210 VJ=100.00  +MOVJ EC00210 VJ=100.00
MOVJ C00211 BC00211 VJ=100.00  +MOVJ EC00211 VJ=100.00
END
